{attribute 'qualified_only'}
{attribute 'strict'}
{attribute 'to_string'}
TYPE E_SnappyVerificationState :
(
	eIdle := 0,
	eSend,
	ePending,
	eDone,
	eError := -1
);
END_TYPE
//  eError = '-1'

(* stored: Version 1.1.0.1, ProductVersion 3.1.4026.18
   EnumerationTextList E_SnappyVerificationState: Id {1e6e5f12-15f0-4500-bf41-d1a982bdf091} *)
